{attribute 'qualified_only'}
VAR_GLOBAL CONSTANT
	// Encoder reference values in counts = nm
	// Enc reference values after alignment 3-13-20
	nYLEFT_ENC_REF : ULINT := 96270560;
	nYRIGHT_ENC_REF : ULINT := 98728200;
	nXUP_ENC_REF : ULINT := 19847200;
	nXDWN_ENC_REF : ULINT := 21007520;
END_VAR

(* stored: Version 1.1.0.1, ProductVersion 3.1.4022.18
   GVL GVL_M1K2_Constants: Id {17631110-39aa-4b3d-a55d-c2ce2a77172f} *)
